PROGRAM JobsExample
VAR
END_VAR

CountToExample();

END_PROGRAM

(* stored: Version 1.1.0.1
   POU JobsExample: Id {10f1f85b-51a8-4846-bc26-10052eed5c0e}, SpecialFunc None *)
